// TIA Portal V17 export
// export: Created 2025-03-07T09:18:55.2051888Z, ExportSetting WithDefaults, DisplayName Totally Integrated Automation Portal, DisplayVersion V17 Update 8, DisplayName TIA Portal Openness, DisplayVersion V17 Update 8, DisplayName TIA Portal Version Control Interface, DisplayVersion V17, DisplayName SINAMICS Startdrive Advanced, DisplayVersion V17 SP2, DisplayName SINAMICS Startdrive G110M, G120, G120C, G120D, G120P, G115D, DisplayVersion V17 SP2, DisplayName SINAMICS Startdrive G130, G150, S120, S150, SINAMICS MV, S210, DisplayVersion V17 SP2, DisplayName STEP 7 Professional, DisplayVersion V17 Update 8, DisplayName SINUMERIK ONE STEP 7 Toolbox, DisplayVersion V17 Update 12, DisplayName SINUMERIK 840D sl STEP 7 Toolbox, DisplayVersion V17 Update 12, DisplayName STEP 7 Safety, DisplayVersion V17 Update 6, DisplayName WinCC Advanced, DisplayVersion V17 Update 8
DATA_BLOCK "DB20231_TRUMPF_LASER_UNIT_02_ACTIVE"   // DB20231
{ DB_Accessible_From_OPC_UA := 'FALSE' }
VERSION : 0.1
// stored: AutoNumber false, DBAccessibleFromOPCUA false, DBAccessibleFromWebserver true, InstanceOfName FB20202_TRUMPF_ACTIVE, InstanceOfType FB
"FB20202_TRUMPF_ACTIVE"
   // VAR_INPUT
   //    iREADY_TO_EMISSION : Bool;
   //    "AIR COMPRESSED OK" : Bool;
   //    iPROGRAM_ACTIVE : Bool;
   //    iExternal_In : Bool;
   //    iMANUAL_START_REQUEST : Bool;
   //    iAUTO_START_REQUEST : Bool;
   //    iMANUAL_STOP_REQUEST : Bool;
   //    iAUTO_STOP_REQUEST : Bool;
   //    iProfile_Enable : Bool;
   //    iStart_Program_Request : Bool;
   //    iUNIT_RESET_LOCAL_SEQ : Bool;
   //    iSAFETY_GATES_CLOSED_LOCKED : Bool;
   //    iPART_PRESENTE : Bool;
   //    iLASER_READY_SC_STATUS : Bool;
   //    iMACHINE_ON_DELAYED : Bool;
   // END_VAR
   // VAR_OUTPUT
   //    oEMISSION_SWITCH_ON : Bool;
   //    oPROGRAM_START : Bool;
   //    oALARM_PROGRAM_NOT_ACTIVE : Bool;
   //    oALARM_NO_LASER_EMISSION : Bool;
   //    oALARM_UNSAFE_STATE : Bool;
   //    oALARM_UNSAFE_AREA : Bool;
   //    "oALARM_LASER-DSS_ANALOG_MODE_MISMATCH" : Bool;
   //    oSTATION_SEOC_ALARMS : Bool;
   // END_VAR
   // VAR RETAIN
   //    DATA : "LASER ACTIVE";
   //    "TIMER FAULT 1" { S7_SetPoint := 'True'} : TON_TIME;
   //    "TIMER FAULT 2" { S7_SetPoint := 'True'} : TON_TIME;
   //    "DELAY EXTERNAL IN" { S7_SetPoint := 'True'} : TON_TIME;
   // END_VAR
BEGIN
END_DATA_BLOCK
